DATA_BLOCK "iFB_Map_Siwarex_Core"
{ S7_Optimized_Access := 'FALSE' }
AUTHOR : S7C_Lib
FAMILY : Analog
VERSION : 1.4
"FB_Map_Siwarex_Core"

BEGIN

END_DATA_BLOCK

